(* IEC 61131-3 sources: conversion/src/strings, 12 files *)

(* ---- ConversionMode.st ---- *)
NAMESPACE Simatic.Ax.Conversion

    /// Represents the conversion mode for integer-to-string operations.
    ///
    /// This type defines the available modes for formatting integer-to-string conversions:
    /// - `NONE`: No special formatting is applied.
    /// - `FORCE_SIGN`: Forces the inclusion of a '+' sign for positive numbers.
    TYPE
        ConversionMode : WORD (NONE := WORD#16#0000, FORCE_SIGN := WORD#16#0001) := NONE;
    END_TYPE

END_NAMESPACE

(* ---- AnyIntToString.st ---- *)
USING System.Strings;
USING System.Math;

NAMESPACE Simatic.Ax.Conversion

    /// Converts a signed 64-bit integer (LINT) to its string representation.
    ///
    /// This function converts a signed 64-bit integer to a string, optionally adding a sign
    /// based on the specified conversion mode. It handles negative values and ensures the
    /// correct number of digits are included in the output.
    ///
    /// @param value The signed 64-bit integer to convert.
    /// @param mode The conversion mode (e.g., force sign).
    /// @return A string representation of the input integer.
    FUNCTION INTERNAL AnyIntToString : STRING
        VAR_INPUT
            value : LINT;
            mode : ConversionMode := ConversionMode#NONE;
        END_VAR
        VAR_TEMP
            _value : LINT;
            digit : INT;
            c : USINT;
            i : INT;
            digits : INT;
            offset : INT;
            s : STRING[1];
            t : ARRAY[0..19] OF CHAR; // MAX: -9223372036854775808
        END_VAR

        _value := value;
        digits := CountDigits(value);
        IF (_value < 0) THEN  // Add sign to
            AnyIntToString := Concat(AnyIntToString, '-');
            offset := 1; // keep space for the sign
        ELSIF (_value > 0 AND (mode AND ConversionMode#FORCE_SIGN) = ConversionMode#FORCE_SIGN) THEN  // Add sign to
            AnyIntToString := Concat(AnyIntToString, '+');
            offset := 1; // keep space for the sign
        ELSE
            offset := 0;
        END_IF;

        FOR i := 0 TO digits - 1 DO
            digit := ABS(TO_INT(_value MOD 10));
            c := TO_USINT('0') + TO_USINT(digit);
            t[digits - i - 1] := TO_CHAR(TO_BYTE(c));
            _value := _value / 10;
        END_FOR;
        FOR i := 0 TO digits - 1 DO
            s[1] := t[i];
            AnyIntToString := Concat(AnyIntToString, s);
        END_FOR;
    END_FUNCTION

    /// Converts an unsigned 64-bit integer (ULINT) to its string representation.
    ///
    /// This function converts an unsigned 64-bit integer to a string, optionally adding a sign
    /// based on the specified conversion mode. It ensures the correct number of digits are
    /// included in the output.
    ///
    /// @param value The unsigned 64-bit integer to convert.
    /// @param mode The conversion mode (e.g., force sign).
    /// @return A string representation of the input integer.
    FUNCTION INTERNAL ULintToString : STRING
        VAR_INPUT
            value : ULINT;
            mode : ConversionMode := ConversionMode#NONE;
        END_VAR
        VAR_TEMP
            _value : ULINT;
            digit : INT;
            c : USINT;
            i : INT;
            digits : INT;
            offset : INT;
            s : STRING[1];
            t : ARRAY[0..19] OF CHAR; // MAX: -9223372036854775808
        END_VAR

        _value := value;
        // Prepare the sting with the correct lenght
        digits := CountDigits(value);

        IF (_value > ULINT#0 AND (mode AND ConversionMode#FORCE_SIGN) = ConversionMode#FORCE_SIGN) THEN  // Add sign to
            ULintToString[1] := '+';
            offset := 1; // keep space for the sign
        ELSE
            offset := 0;
        END_IF;

        FOR i := 0 TO digits - 1 DO
            digit := ABS(TO_INT(_value MOD UINT#10));
            c := TO_USINT('0') + TO_USINT(digit);
            t[digits - i - 1] := TO_CHAR(TO_BYTE(c));
            _value := _value / UINT#10;
        END_FOR;
        FOR i := 0 TO digits - 1 DO
            s[1] := t[i];
            ULintToString := Concat(ULintToString, s);
        END_FOR;
    END_FUNCTION

END_NAMESPACE

(* ---- ArrayToString.st ---- *)
USING System.Strings;

NAMESPACE Simatic.Ax.Conversion.Arrays

    /// Converts a subset of a character array to a string.
    ///
    /// This function takes a character array and converts a specified range of elements
    /// (from `startIdx` to `endIdx`) into a string. If the range is invalid or exceeds
    /// the array bounds, an empty string is returned. The maximum string length is limited
    /// to `MAX_STR_LEN`.
    ///
    /// @param arr The input character array.
    /// @param startIdx The starting index of the range to convert.
    /// @param endIdx The ending index of the range to convert.
    /// @return A string representation of the specified range of the array.
    {axcode:docs-v0:@simatic-ax/conversion:ArrayToString.md}
    FUNCTION ToString : STRING
        VAR_INPUT
            arr : ARRAY[*] OF CHAR;
            startIdx : INT;
            endIdx : INT;
        END_VAR
        VAR CONSTANT
            MAX_STR_LEN : INT := 254;
        END_VAR
        VAR_TEMP
            i : DINT;
            _lb : DINT;
            _ub : DINT;
            _arrayLen : DINT;
        END_VAR
        _lb := LOWER_BOUND(arr, 1);
        _ub := UPPER_BOUND(arr, 1);

        // start index > end index
        IF (startIdx > endIdx) THEN
            ToString := '';
            RETURN;
        END_IF;

        // start index is not existing
        IF (startIdx < _lb) OR (startIdx > _ub) AND (startIdx <> 0) THEN
            ToString := '';
            RETURN;
        END_IF;
        // end index is ot existing
        IF (endIdx > _ub) THEN
            ToString := '';
            RETURN;
        END_IF;
        _arrayLen := endIdx - startIdx + 1;

        IF (_arrayLen > MAX_STR_LEN) THEN
            _arrayLen := MAX_STR_LEN;
        END_IF;

        FOR i := 0 TO _arrayLen - 1 DO
            ToString[i + 1] := arr[i + _lb + startIdx];
        END_FOR;

    END_FUNCTION

    /// Converts an entire character array to a string.
    ///
    /// This function takes a character array and converts all its elements into a string.
    /// If the array length exceeds `MAX_STR_LEN`, the resulting string is truncated to
    /// the maximum allowed length.
    ///
    /// @param arr The input character array.
    /// @return A string representation of the entire array.
    {axcode:docs-v0:@simatic-ax/conversion:ArrayToString.md}
    FUNCTION ToString : STRING
        VAR_INPUT
            arr : ARRAY[*] OF CHAR;
        END_VAR
        VAR CONSTANT
            MAX_STR_LEN : INT := 254;
        END_VAR
        VAR_TEMP
            i : DINT;
            _lb : DINT;
            _ub : DINT;
            _arrayLen : DINT;
        END_VAR
        _lb := LOWER_BOUND(arr, 1);
        _ub := UPPER_BOUND(arr, 1);

        _arrayLen := _ub - _lb + 1;

        IF (_arrayLen > MAX_STR_LEN) THEN
            _arrayLen := MAX_STR_LEN;
        END_IF;

        FOR i := 0 TO _arrayLen - 1 DO
            ToString[i + 1] := arr[i + _lb];
        END_FOR;

    END_FUNCTION

END_NAMESPACE

(* ---- CountDigits.st ---- *)
NAMESPACE Simatic.Ax.Conversion

    /// Counts the number of digits in a signed 64-bit integer (LINT).
    ///
    /// This function calculates the number of decimal digits in the given signed 64-bit integer.
    /// It iteratively checks the range of the value against increasing powers of 10.
    /// The maximum number of digits it can handle is defined by `MAX_DIGITS`.
    ///
    /// @param value The signed 64-bit integer whose digits are to be counted.
    /// @return The number of decimal digits in the input value.
    {axcode:docs-v0:@simatic-ax/conversion:CountDigits.md}
    FUNCTION CountDigits : INT
        VAR_INPUT
            value : LINT;
        END_VAR
        VAR_TEMP
            divisor : LINT := LINT#10;
            i : INT;
        END_VAR
        VAR CONSTANT
            MAX_DIGITS : INT := 18;
        END_VAR

        FOR i := 1 TO MAX_DIGITS DO
            IF((value > (LINT#-1 * divisor)) AND (value < divisor)) THEN
                CountDigits := i;
                RETURN;
            END_IF;
            divisor := divisor * LINT#10;
        END_FOR;
        CountDigits := 19;
    END_FUNCTION

    /// Counts the number of digits in an unsigned 64-bit integer (ULINT).
    ///
    /// This function calculates the number of decimal digits in the given unsigned 64-bit integer.
    /// It iteratively checks the range of the value against increasing powers of 10.
    /// The maximum number of digits it can handle is defined by `MAX_DIGITS`.
    ///
    /// @param value The unsigned 64-bit integer whose digits are to be counted.
    /// @return The number of decimal digits in the input value.
    {axcode:docs-v0:@simatic-ax/conversion:CountDigits.md}
    FUNCTION CountDigits : INT
        VAR_INPUT
            value : ULINT;
        END_VAR
        VAR_TEMP
            divisor : ULINT := ULINT#10;
            i : INT;
        END_VAR
        VAR CONSTANT
            MAX_DIGITS : INT := 19;
        END_VAR

        FOR i := 1 TO MAX_DIGITS DO
            IF(value < divisor) THEN
                CountDigits := i;
                RETURN;
            END_IF;
            divisor := divisor * UINT#10;
        END_FOR;
        CountDigits := 20;
    END_FUNCTION

END_NAMESPACE

(* ---- HexToString.st ---- *)
USING System;
USING System.Strings;

NAMESPACE Simatic.Ax.Conversion

    /// Converts a BYTE value to its hexadecimal string representation.
    ///
    /// This function takes a BYTE value and converts it into a two-character hexadecimal string.
    /// It splits the BYTE into two nibbles, converts each nibble to its hexadecimal character,
    /// and concatenates the results.
    ///
    /// @param b The BYTE value to convert.
    /// @return A two-character string representing the hexadecimal value of the input BYTE.
    {axcode:docs-v0:@simatic-ax/conversion:HexToString.md}
    FUNCTION PUBLIC ByteToString : STRING
        VAR_INPUT
            b : BYTE;
        END_VAR
        VAR_TEMP
            tempN1 : BYTE;
            tempN2 : BYTE;
        END_VAR
        tempN1 := b AND BYTE#16#0F;
        tempN2 := SHR(b,USINT#4);

        ByteToString := Concat(LookUpHEX(tempN2),LookUpHEX(tempN1));

    END_FUNCTION

    /// Converts a nibble (4 bits) to its hexadecimal character representation.
    ///
    /// This function takes a nibble (a value between 0 and 15) and returns the corresponding
    /// hexadecimal character (0-9, A-F) using a lookup table.
    ///
    /// @param nibble The nibble value to convert (0-15).
    /// @return The hexadecimal character corresponding to the input nibble.
    FUNCTION INTERNAL LookUpHEX : CHAR
        VAR_INPUT
            nibble : BYTE;
        END_VAR
        VAR
            h : ARRAY[0..15] of CHAR := ['0','1','2','3','4','5','6','7','8','9','A','B','C','D','E','F'];
        END_VAR

        LookUpHEX := h[TO_UINT(nibble)];

    END_FUNCTION

END_NAMESPACE

(* ---- IntToString.st ---- *)
USING System.Strings;

NAMESPACE Simatic.Ax.Conversion.Integer

    /// Converts a signed 8-bit integer (SINT) to a string.
    ///
    /// This function converts a signed 8-bit integer to its string representation.
    /// The conversion supports an optional mode parameter to customize the output format.
    ///
    /// @param value The signed 8-bit integer to convert.
    /// @param mode The conversion mode (e.g., force sign).
    /// @return A string representation of the input integer.
    {axcode:docs-v0:@simatic-ax/conversion:IntToString.md}
    FUNCTION ToString : STRING[4]
        VAR_INPUT
            value : SINT;
            mode : ConversionMode := ConversionMode#NONE;
        END_VAR
        VAR_TEMP
        END_VAR
        ToString := AnyIntToString(value := value, mode := mode);
    END_FUNCTION

    /// Converts an unsigned 8-bit integer (USINT) to a string.
    ///
    /// This function converts an unsigned 8-bit integer to its string representation.
    /// The conversion supports an optional mode parameter to customize the output format.
    ///
    /// @param value The unsigned 8-bit integer to convert.
    /// @param mode The conversion mode (e.g., force sign).
    /// @return A string representation of the input integer.
    {axcode:docs-v0:@simatic-ax/conversion:IntToString.md}
    FUNCTION ToString : STRING[4]
        VAR_INPUT
            value : USINT;
            mode : ConversionMode := ConversionMode#NONE;
        END_VAR
        VAR_TEMP
        END_VAR
        ToString := AnyIntToString(value := value, mode := mode);
    END_FUNCTION

    /// Converts a signed 16-bit integer (INT) to a string.
    ///
    /// This function converts a signed 16-bit integer to its string representation.
    /// The conversion supports an optional mode parameter to customize the output format.
    ///
    /// @param value The signed 16-bit integer to convert.
    /// @param mode The conversion mode (e.g., force sign).
    /// @return A string representation of the input integer.
    {axcode:docs-v0:@simatic-ax/conversion:IntToString.md}
    FUNCTION ToString : STRING[6]
        VAR_INPUT
            value : INT;
            mode : ConversionMode := ConversionMode#NONE;
        END_VAR
        VAR_TEMP
        END_VAR
        ToString := AnyIntToString(value := value, mode := mode);
    END_FUNCTION

    /// Converts an unsigned 16-bit integer (UINT) to a string.
    ///
    /// This function converts an unsigned 16-bit integer to its string representation.
    /// The conversion supports an optional mode parameter to customize the output format.
    ///
    /// @param value The unsigned 16-bit integer to convert.
    /// @param mode The conversion mode (e.g., force sign).
    /// @return A string representation of the input integer.
    {axcode:docs-v0:@simatic-ax/conversion:IntToString.md}
    FUNCTION ToString : STRING[6]
        VAR_INPUT
            value : UINT;
            mode : ConversionMode := ConversionMode#NONE;
        END_VAR
        VAR_TEMP
        END_VAR
        ToString := AnyIntToString(value := value, mode := mode);
    END_FUNCTION

    /// Converts a signed 32-bit integer (DINT) to a string.
    ///
    /// This function converts a signed 32-bit integer to its string representation.
    /// The conversion supports an optional mode parameter to customize the output format.
    ///
    /// @param value The signed 32-bit integer to convert.
    /// @param mode The conversion mode (e.g., force sign).
    /// @return A string representation of the input integer.
    {axcode:docs-v0:@simatic-ax/conversion:IntToString.md}
    FUNCTION ToString : STRING[11]
        VAR_INPUT
            value : DINT;
            mode : ConversionMode := ConversionMode#NONE;
        END_VAR
        VAR_TEMP
        END_VAR
        ToString := AnyIntToString(value := value, mode := mode);
    END_FUNCTION

    /// Converts an unsigned 32-bit integer (UDINT) to a string.
    ///
    /// This function converts an unsigned 32-bit integer to its string representation.
    /// The conversion supports an optional mode parameter to customize the output format.
    ///
    /// @param value The unsigned 32-bit integer to convert.
    /// @param mode The conversion mode (e.g., force sign).
    /// @return A string representation of the input integer.
    {axcode:docs-v0:@simatic-ax/conversion:IntToString.md}
    FUNCTION ToString : STRING[11]
        VAR_INPUT
            value : UDINT;
            mode : ConversionMode := ConversionMode#NONE;
        END_VAR
        VAR_TEMP
        END_VAR
        ToString := AnyIntToString(value := value, mode := mode);
    END_FUNCTION

    /// Converts a signed 64-bit integer (LINT) to a string.
    ///
    /// This function converts a signed 64-bit integer to its string representation.
    /// The conversion supports an optional mode parameter to customize the output format.
    ///
    /// @param value The signed 64-bit integer to convert.
    /// @param mode The conversion mode (e.g., force sign).
    /// @return A string representation of the input integer.
    {axcode:docs-v0:@simatic-ax/conversion:IntToString.md}
    FUNCTION ToString : STRING[20]
        VAR_INPUT
            value : LINT;
            mode : ConversionMode := ConversionMode#NONE;
        END_VAR
        VAR_TEMP
        END_VAR
        ToString := AnyIntToString(value := value, mode := mode);
    END_FUNCTION

    /// Converts an unsigned 64-bit integer (ULINT) to a string.
    ///
    /// This function converts an unsigned 64-bit integer to its string representation.
    /// The conversion supports an optional mode parameter to customize the output format.
    ///
    /// @param value The unsigned 64-bit integer to convert.
    /// @param mode The conversion mode (e.g., force sign).
    /// @return A string representation of the input integer.
    {axcode:docs-v0:@simatic-ax/conversion:IntToString.md}
    FUNCTION ToString : STRING[21]
        VAR_INPUT
            value : ULINT;
            mode : ConversionMode := ConversionMode#NONE;
        END_VAR
        VAR_TEMP
        END_VAR
        ToString := ULintToString(value := value, mode := mode);
    END_FUNCTION

END_NAMESPACE

(* ---- StringToAnyInt.st ---- *)
USING System.Strings;

NAMESPACE Simatic.Ax.Conversion

    /// Converts a string to a signed 64-bit integer (LINT).
    ///
    /// This function parses a string and converts it to a signed 64-bit integer. It handles
    /// optional '+' or '-' signs and checks for overflow. If the string is invalid, the
    /// function returns FALSE and sets the output to 0.
    ///
    /// @param str The input string to convert.
    /// @return TRUE if the conversion is successful, FALSE otherwise.
    {axcode:docs-v0:@simatic-ax/conversion:StringToAnyInt.md}
    FUNCTION StringToAnyInt : BOOL
        VAR_INPUT
            str : STRING;
        END_VAR
        VAR_OUTPUT
            value : LINT;
        END_VAR
        VAR_TEMP
            _len : INT;
            i : INT;
            _val : INT;
            _val_max : INT;
            _sig : INT;
            _start : INT;
            _c : STRING;
        END_VAR

        _len := LengthOf(str);

        IF (str[1] = '+') THEN
            _sig := 1;
            _start := 2;
            _val_max := 7; // = 2^63-1 MOD 10
        ELSIF (str[1] = '-') THEN
            _sig := -1;
            _start := 2;
            _val_max := 8; // = 2^63   MOD 10
        ELSE
            _sig := 1;
            _start := 1;
            _val_max := 7; // = 2^63-1 MOD 10
        END_IF;

        value := 0;

        IF (_len - _start < 0) THEN
            // no digits.
            StringToAnyInt := FALSE;
            RETURN;
        END_IF;

        FOR i := _start TO _len DO
            _c := str[i];
            CASE _c OF
                '0' : _val := 0;
                '1' : _val := 1;
                '2' : _val := 2;
                '3' : _val := 3;
                '4' : _val := 4;
                '5' : _val := 5;
                '6' : _val := 6;
                '7' : _val := 7;
                '8' : _val := 8;
                '9' : _val := 9;
            ELSE
                value := 0;
                StringToAnyInt := FALSE;
                RETURN;
            END_CASE;

            IF ((value < 0) OR //previously accepted overflow for minimum of LINT
                // 2^63-1    >9223372036854775807
                (value > LINT#922337203685477580) OR
                (value = LINT#922337203685477580 AND _val > _val_max)) THEN
                // overflow
                value := LINT#0;
                StringToAnyInt := FALSE;
                RETURN;
            END_IF;

            value := value * 10;
            value := value + _val;
        END_FOR;
        value := value * _sig;

        StringToAnyInt := TRUE;

    END_FUNCTION

    /// Converts a string to an unsigned 64-bit integer (ULINT).
    ///
    /// This function parses a string and converts it to an unsigned 64-bit integer. It handles
    /// optional '+' signs and checks for overflow. If the string is invalid, the function
    /// returns FALSE and sets the output to 0.
    ///
    /// @param str The input string to convert.
    /// @return TRUE if the conversion is successful, FALSE otherwise.
    FUNCTION INTERNAL StringToULint: BOOL
        VAR_INPUT
            str : STRING;
        END_VAR
        VAR_OUTPUT
            value : ULINT;
        END_VAR
        VAR_TEMP
            _len : INT;
            i : INT;
            _val : ULINT;
            _start : INT;
            _c : STRING;
        END_VAR

        _len := LengthOf(str);

        IF (str[1] = '+') THEN
            _start := 2;
        ELSE
            _start := 1;
        END_IF;

        value := ULINT#0;

        IF (_len - _start < 0) THEN
            // no digits.
            StringToULint := FALSE;
            RETURN;
        END_IF;

        FOR i := _start TO _len DO

            _c := str[i];
            CASE _c OF
                '0' : _val := ULINT#0;
                '1' : _val := ULINT#1;
                '2' : _val := ULINT#2;
                '3' : _val := ULINT#3;
                '4' : _val := ULINT#4;
                '5' : _val := ULINT#5;
                '6' : _val := ULINT#6;
                '7' : _val := ULINT#7;
                '8' : _val := ULINT#8;
                '9' : _val := ULINT#9;
            ELSE
                value := ULINT#0;
                StringToULint := FALSE;
                RETURN;
            END_CASE;

            IF ((value > ULINT#1844674407370955161) OR (value = ULINT#1844674407370955161 AND _val > ULINT#5)) THEN
                //  2^64 - 1 = 18446744073709551616
                // overflow
                value := ULINT#0;
                StringToULint := FALSE;
                RETURN;
            END_IF;

            value := value * ULINT#10;
            value := value + _val;
        END_FOR;
        StringToULint := TRUE;
    END_FUNCTION

END_NAMESPACE

(* ---- StringToArrayOfCharCount.st ---- *)
USING System.Strings;

NAMESPACE Simatic.Ax.Conversion.Strings.ToArray

    /// Converts a string to an array of CHAR values.
    ///
    /// This function copies characters from the input string into the provided array of CHAR.
    /// It returns the number of characters copied. If the array is smaller than the string,
    /// the output is truncated to fit the array size.
    ///
    /// @param str The input string to convert.
    /// @param arr The output array to store the CHAR values.
    /// @return The number of characters copied to the array.
    {axcode:docs-v0:@simatic-ax/conversion:StringToArrayOfCharCount.md}
    FUNCTION OfCharCount : DINT
        VAR_INPUT
            str : STRING;
        END_VAR
        VAR_IN_OUT
            arr : ARRAY[*] OF CHAR;
        END_VAR
        VAR_TEMP
            i : DINT;
            _lb : DINT;
            _ub : DINT;
            _maxLen : DINT;
        END_VAR
        _lb := LOWER_BOUND(arr, 1);
        _ub := UPPER_BOUND(arr, 1);
        _maxLen := LengthOf(str);

        IF (_maxLen > _ub - _lb + 1) THEN
            _maxLen := TO_INT(_ub - _lb + 1);
        END_IF;

        FOR i := 0 TO _maxLen - 1 DO
            arr[i + _lb] := str[i + 1];
        END_FOR;
        OfCharCount := i;
    END_FUNCTION

END_NAMESPACE

(* ---- StringToArrayOfLint.st ---- *)
USING Simatic.Ax.Conversion.Strings;
USING System.Strings;

NAMESPACE Simatic.Ax.Conversion.Strings.ToArray

    /// Converts a string representation of an array of integers to an array of LINT values.
    ///
    /// This function parses a string containing integers (e.g., "[1, 2, 3]") and converts it
    /// into an array of LINT values. If the string cannot be converted, the function returns FALSE.
    ///
    /// @param str The input string to parse.
    /// @param arr The output array to store the converted LINT values.
    /// @return TRUE if the conversion is successful, FALSE otherwise.
    FUNCTION INTERNAL OfLint : BOOL
        VAR_INPUT
            str: STRING;
        END_VAR
        VAR_IN_OUT
            arr: ARRAY[*] OF LINT;
        END_VAR
        VAR_TEMP
            arrayStart: INT;
            arrayEnd: INT;
            lb: DINT;
            ub: DINT;
            index: INT;
            intString: STRING;
            arrayIndex: DINT;

            elementStart: INT;
            elementEnd: INT;
            inElement: BOOL := FALSE;
            elementFound: BOOL := FALSE;
            ch : CHAR;
            substr: STRING;
            parseSucces: BOOL;

            value: LINT; //mehr möglich machen!
        END_VAR

        OfLint := FALSE;
        IF LengthOf(str) = 0 THEN
            RETURN;
        END_IF;

        lb := LOWER_BOUND(arr, 1);
        ub := UPPER_BOUND(arr, 1);

        GetArrayBounds(str, arrayStart, arrayEnd);

        arrayIndex := LOWER_BOUND(arr, 1);
        //loop through string
        FOR index := arrayStart TO arrayEnd DO

            ch := str[index];

            IF (NOT inElement AND ch = ']') THEN
                OfLint := TRUE;
                RETURN;
            END_IF;

            IF NOT inElement AND NOT ((ch = ' ' OR ch = ',')) THEN
                elementStart := index;
                inElement := TRUE;
            END_IF;

            IF inElement AND (ch = ' ' OR ch = ',' OR ch = ']') THEN
                elementEnd := index;
                inElement := FALSE;
                elementFound := TRUE;
            END_IF;

            IF elementFound THEN

                substr := Substring(str, elementStart, elementEnd - elementStart);
                parseSucces := StringToAnyInt(substr, value);

                IF parseSucces THEN
                    IF (arrayIndex > ub) THEN
                        OfLint := TRUE;
                        RETURN;
                    END_IF;
                    arr[arrayIndex] := value;
                    OfLint := TRUE;
                    arrayIndex := arrayIndex + 1;
                    elementFound := FALSE;
                ELSE
                    OfLint := FALSE;
                    RETURN;
                END_IF;
            END_IF;
        END_FOR;
    END_FUNCTION

    /// Extracts the bounds of an array from a string representation.
    ///
    /// This function identifies the positions of the opening and closing brackets
    /// in a string representing an array (e.g., "[1, 2, 3]") and returns their indices.
    ///
    /// @param str The input string to analyze.
    /// @param lower The index of the opening bracket.
    /// @param upper The index of the closing bracket.
    {axcode:docs-v0:@simatic-ax/conversion:StringToArrayOfLint.md}
    FUNCTION GetArrayBounds
        VAR_INPUT
            str: STRING;
        END_VAR
        VAR_OUTPUT
            lower: INT;
            upper: INT;
        END_VAR
        VAR
            index: INT;
        END_VAR

        FOR index := 1 TO LengthOf(str) DO
            IF str[index] = '[' THEN
                lower := index + 1;
                EXIT;
            END_IF;
        END_FOR;

        FOR index := LengthOf(str) TO 1 BY -1 DO
            IF str[index] = ']' THEN
                upper := index;
                EXIT;
            END_IF;
        END_FOR;

    END_FUNCTION

END_NAMESPACE

(* ---- StringToArrayOfLintCount.st ---- *)
USING Simatic.Ax.Conversion.Strings;
USING System.Strings;

NAMESPACE Simatic.Ax.Conversion.Strings.ToArray

    /// Converts a string representation of an array of integers to an array of LINT values.
    ///
    /// This function parses a string containing integers (e.g., "[1, 2, 3]") and converts it
    /// into an array of LINT values. It returns the number of successfully converted elements.
    /// If the string cannot be converted, the function returns 0.
    ///
    /// @param str The input string to parse.
    /// @param arr The output array to store the converted LINT values.
    /// @return The number of successfully converted elements.
    FUNCTION INTERNAL OfLintCount : DINT
        VAR_INPUT
            str: STRING;
        END_VAR
        VAR_IN_OUT
            arr: ARRAY[*] OF LINT;
        END_VAR
        VAR_TEMP
            arrayStart: INT;
            arrayEnd: INT;
            lb: DINT;
            ub: DINT;
            index: INT;
            intString: STRING;
            arrayIndex: DINT;
            count: DINT;

            elementStart: INT;
            elementEnd: INT;
            inElement: BOOL := FALSE;
            elementFound: BOOL := FALSE;
            ch : CHAR;
            substr: STRING;
            parseSucces: BOOL;

            value: LINT; //mehr möglich machen!
        END_VAR

        OfLintCount := 0;
        IF LengthOf(str) = 0 THEN
            RETURN;
        END_IF;

        lb := LOWER_BOUND(arr, 1);
        ub := UPPER_BOUND(arr, 1);

        GetArrayBounds(str, arrayStart, arrayEnd);

        arrayIndex := LOWER_BOUND(arr, 1);
        //loop through string
        FOR index := arrayStart TO arrayEnd DO

            ch := str[index];

            IF (NOT inElement AND ch = ']') THEN
                OfLintCount := count;
                RETURN;
            END_IF;

            IF NOT inElement AND NOT ((ch = ' ' OR ch = ',')) THEN
                elementStart := index;
                inElement := TRUE;
            END_IF;

            IF inElement AND (ch = ' ' OR ch = ',' OR ch = ']') THEN
                elementEnd := index;
                inElement := FALSE;
                elementFound := TRUE;
            END_IF;

            IF elementFound THEN

                substr := Substring(str, elementStart, elementEnd - elementStart);
                parseSucces := StringToAnyInt(substr, value);

                IF parseSucces THEN
                    IF (arrayIndex > ub) THEN
                        OfLintCount := count;
                        RETURN;
                    END_IF;
                    arr[arrayIndex] := value;
                    count := count + 1;
                    OfLintCount := count;
                    arrayIndex := arrayIndex + 1;
                    elementFound := FALSE;
                ELSE
                    OfLintCount := 0;
                    RETURN;
                END_IF;
            END_IF;
        END_FOR;
    END_FUNCTION

END_NAMESPACE

(* ---- StringToBool.st ---- *)
USING Simatic.Ax.Conversion.Strings;
USING System.Strings;

NAMESPACE Simatic.Ax.Conversion

    /// Converts a string to a boolean value.
    ///
    /// This function checks if the input string represents "TRUE" or "FALSE" (case-insensitive).
    /// If the string matches "TRUE", the output is TRUE. If it matches "FALSE", the output is FALSE.
    /// Otherwise, the function returns FALSE and sets the output to FALSE.
    ///
    /// @param str The input string to convert.
    /// @return TRUE if the conversion is successful, FALSE otherwise.
    {axcode:docs-v0:@simatic-ax/conversion:StringToBool.md}
    FUNCTION StringToBool : BOOL
        VAR_INPUT
            str: STRING;
        END_VAR
        VAR_OUTPUT
            value: BOOL;
        END_VAR

        IF LengthOf(str) < 4 OR LengthOf(str) > 5 THEN
            value:= FALSE; StringToBool := FALSE;
            RETURN;
        END_IF;

        IF LengthOf(str) = 5 THEN
            IF NOT (str[1] = 'F' OR str[1] = 'f') THEN
                StringToBool := FALSE;
                RETURN;
            END_IF;
            IF NOT (str[2] = 'A' OR str[2] = 'a') THEN
                StringToBool := FALSE;
                RETURN;
            END_IF;
            IF NOT (str[3] = 'L' OR str[3] = 'l') THEN
                StringToBool := FALSE;
                RETURN;
            END_IF;
            IF NOT (str[4] = 'S' OR str[4] = 's') THEN
                StringToBool := FALSE;
                RETURN;
            END_IF;
            IF NOT (str[5] = 'E' OR str[5] = 'e') THEN
                StringToBool := FALSE;
                RETURN;
            END_IF;
            value:= FALSE;
            StringToBool := TRUE;
            RETURN;
        END_IF;

        IF LengthOf(str) = 4 THEN
            IF NOT (str[1] = 'T' OR str[1] = 't') THEN
                StringToBool := FALSE;
                RETURN;
            END_IF;
            IF NOT (str[2] = 'R' OR str[2] = 'r') THEN
                StringToBool := FALSE;
                RETURN;
            END_IF;
            IF NOT (str[3] = 'U' OR str[3] = 'u') THEN
                StringToBool := FALSE;
                RETURN;
            END_IF;
            IF NOT (str[4] = 'E' OR str[4] = 'e') THEN
                StringToBool := FALSE;
                RETURN;
            END_IF;
            value:= TRUE;
            StringToBool := TRUE;
        END_IF;
    END_FUNCTION

END_NAMESPACE

(* ---- ToInt.st ---- *)
USING System.Strings;

NAMESPACE Simatic.Ax.Conversion.Strings

    /// Converts a string to a signed 8-bit integer (SINT).
    ///
    /// This function parses a string and converts it to a signed 8-bit integer. If the value
    /// is out of range or invalid, the function returns FALSE and sets the output to 0.
    ///
    /// @param str The input string to convert.
    /// @return TRUE if the conversion is successful, FALSE otherwise.
    {axcode:docs-v0:@simatic-ax/conversion:ToInt.md}
    FUNCTION ToInt : BOOL
        VAR_INPUT
            str : STRING;
        END_VAR
        VAR_OUTPUT
            value : SINT;
        END_VAR
        VAR_TEMP
            _val : LINT;
        END_VAR
        VAR CONSTANT
            MAX_VAL : LINT := LINT#127;
            MIN_VAL : LINT := LINT#-128;
        END_VAR

        ToInt := StringToAnyInt(str := str, value => _val);

        IF (_val < MIN_VAL) OR (_val > MAX_VAL) THEN
            value := SINT#0;
            ToInt := FALSE;
        ELSE
            value := TO_SINT(_val);
        END_IF;
    END_FUNCTION

    /// Converts a string to a signed 16-bit integer (INT).
    ///
    /// This function parses a string and converts it to a signed 16-bit integer. If the value
    /// is out of range or invalid, the function returns FALSE and sets the output to 0.
    ///
    /// @param str The input string to convert.
    /// @return TRUE if the conversion is successful, FALSE otherwise.
    {axcode:docs-v0:@simatic-ax/conversion:ToInt.md}
    FUNCTION ToInt : BOOL
        VAR_INPUT
            str : STRING;
        END_VAR
        VAR_OUTPUT
            value : INT;
        END_VAR
        VAR_TEMP
            _val : LINT;
        END_VAR
        VAR CONSTANT
            MAX_VAL : LINT := LINT#32767;
            MIN_VAL : LINT := LINT#-32768;
        END_VAR

        ToInt := StringToAnyInt(str := str, value => _val);

        IF (_val < MIN_VAL) OR (_val > MAX_VAL) THEN
            value := SINT#0;
            ToInt := FALSE;
        ELSE
            value := TO_INT(_val);
        END_IF;
    END_FUNCTION

    /// Converts a string to a signed 32-bit integer (DINT).
    ///
    /// This function parses a string and converts it to a signed 32-bit integer. If the value
    /// is out of range or invalid, the function returns FALSE and sets the output to 0.
    ///
    /// @param str The input string to convert.
    /// @return TRUE if the conversion is successful, FALSE otherwise.
    {axcode:docs-v0:@simatic-ax/conversion:ToInt.md}
    FUNCTION ToInt : BOOL
        VAR_INPUT
            str : STRING;
        END_VAR
        VAR_OUTPUT
            value : DINT;
        END_VAR
        VAR_TEMP
            _val : LINT;
        END_VAR
        VAR CONSTANT
            MAX_VAL : LINT := LINT#2147483647;
            MIN_VAL : LINT := LINT#-2147483648;
        END_VAR

        ToInt := StringToAnyInt(str := str, value => _val);

        IF (_val < MIN_VAL) OR (_val > MAX_VAL) THEN
            value := SINT#0;
            ToInt := FALSE;
        ELSE
            value := TO_DINT(_val);
        END_IF;
    END_FUNCTION

    /// Converts a string to a signed 64-bit integer (LINT).
    ///
    /// This function parses a string and converts it to a signed 64-bit integer. If the value
    /// is out of range or invalid, the function returns FALSE and sets the output to 0.
    ///
    /// @param str The input string to convert.
    /// @return TRUE if the conversion is successful, FALSE otherwise.
    {axcode:docs-v0:@simatic-ax/conversion:ToInt.md}
    FUNCTION ToInt : BOOL
        VAR_INPUT
            str : STRING;
        END_VAR
        VAR_OUTPUT
            value : LINT;
        END_VAR
        VAR_TEMP
            _val : LINT;
        END_VAR
        VAR CONSTANT
            MAX_VAL : LINT := LINT#9223372036854775807;
            MIN_VAL : LINT := LINT#-9223372036854775808;
        END_VAR

        ToInt := StringToAnyInt(str := str, value => _val);

        IF (_val < MIN_VAL) OR (_val > MAX_VAL) THEN
            value := SINT#0;
            ToInt := FALSE;
        ELSE
            value := _val;
        END_IF;
    END_FUNCTION

    /// Converts a string to an unsigned 8-bit integer (USINT).
    ///
    /// This function parses a string and converts it to an unsigned 8-bit integer. If the value
    /// is out of range or invalid, the function returns FALSE and sets the output to 0.
    ///
    /// @param str The input string to convert.
    /// @return TRUE if the conversion is successful, FALSE otherwise.
    {axcode:docs-v0:@simatic-ax/conversion:ToInt.md}
    FUNCTION ToInt : BOOL
        VAR_INPUT
            str : STRING;
        END_VAR
        VAR_OUTPUT
            value : USINT;
        END_VAR
        VAR_TEMP
            _val : LINT;
        END_VAR
        VAR CONSTANT
            MAX_VAL : LINT := LINT#255;
            MIN_VAL : LINT := LINT#0;
        END_VAR

        ToInt := StringToAnyInt(str := str, value => _val);

        IF (_val < MIN_VAL) OR (_val > MAX_VAL) THEN
            value := USINT#0;
            ToInt := FALSE;
        ELSE
            value := TO_USINT(_val);
        END_IF;
    END_FUNCTION

    /// Converts a string to an unsigned 16-bit integer (UINT).
    ///
    /// This function parses a string and converts it to an unsigned 16-bit integer. If the value
    /// is out of range or invalid, the function returns FALSE and sets the output to 0.
    ///
    /// @param str The input string to convert.
    /// @return TRUE if the conversion is successful, FALSE otherwise.
    {axcode:docs-v0:@simatic-ax/conversion:ToInt.md}
    FUNCTION ToInt : BOOL
        VAR_INPUT
            str : STRING;
        END_VAR
        VAR_OUTPUT
            value : UINT;
        END_VAR
        VAR_TEMP
            _val : LINT;
        END_VAR
        VAR CONSTANT
            MAX_VAL : LINT := LINT#65535;
            MIN_VAL : LINT := LINT#0;
        END_VAR

        ToInt := StringToAnyInt(str := str, value => _val);

        IF (_val < MIN_VAL) OR (_val > MAX_VAL) THEN
            value := USINT#0;
            ToInt := FALSE;
        ELSE
            value := TO_UINT(_val);
        END_IF;
    END_FUNCTION

    /// Converts a string to an unsigned 32-bit integer (UDINT).
    ///
    /// This function parses a string and converts it to an unsigned 32-bit integer. If the value
    /// is out of range or invalid, the function returns FALSE and sets the output to 0.
    ///
    /// @param str The input string to convert.
    /// @return TRUE if the conversion is successful, FALSE otherwise.
    {axcode:docs-v0:@simatic-ax/conversion:ToInt.md}
    FUNCTION ToInt : BOOL
        VAR_INPUT
            str : STRING;
        END_VAR
        VAR_OUTPUT
            value : UDINT;
        END_VAR
        VAR_TEMP
            _val : LINT;
        END_VAR
        VAR CONSTANT
            MAX_VAL : LINT := LINT#4294967295;
            MIN_VAL : LINT := LINT#0;
        END_VAR

        ToInt := StringToAnyInt(str := str, value => _val);

        IF (_val < MIN_VAL) OR (_val > MAX_VAL) THEN
            value := USINT#0;
            ToInt := FALSE;
        ELSE
            value := TO_UDINT(_val);
        END_IF;
    END_FUNCTION

    /// Converts a string to an unsigned 64-bit integer (ULINT).
    ///
    /// This function parses a string and converts it to an unsigned 64-bit integer. If the value
    /// is out of range or invalid, the function returns FALSE and sets the output to 0.
    ///
    /// @param str The input string to convert.
    /// @return TRUE if the conversion is successful, FALSE otherwise.
    {axcode:docs-v0:@simatic-ax/conversion:ToInt.md}
    FUNCTION ToInt : BOOL
        VAR_INPUT
            str : STRING;
        END_VAR
        VAR_OUTPUT
            value : ULINT;
        END_VAR
        VAR_TEMP
            _val : ULINT;
        END_VAR
        VAR CONSTANT
            MAX_VAL : ULINT := ULINT#18446744073709551615;
            MIN_VAL : ULINT := ULINT#0;
        END_VAR

        ToInt := StringToULint(str := str, value => _val);

        IF (_val < MIN_VAL) OR (_val > MAX_VAL) THEN
            value := USINT#0;
            ToInt := FALSE;
        ELSE
            value := _val;
        END_IF;
    END_FUNCTION

END_NAMESPACE
